FUNCTION TryConvert_INT_TO_INT : BOOL
VAR_INPUT
	in : INT;
	out : REFERENCE TO INT;
END_VAR

out := in;
TryConvert_INT_TO_INT := TRUE;

END_FUNCTION

(* stored: Version 1.1.0.1, ProductVersion 3.1.4024.12
   POU TryConvert_INT_TO_INT: Id {4d7cac21-5b9a-48d0-bfaf-6e725e8777e8}, SpecialFunc None *)
